/// container for all data that are used by the unit
TYPE HandlingDataRef :
STRUCT
  Config : REFERENCE TO HandlingDataConfig; // data required for booting the unit (axes configuration, simulation, parameters that have to be written in PREOP, ...)
  Machine : REFERENCE TO HandlingDataMachine; // speeds, positions, ...
  Calibration : REFERENCE TO HandlingDataCalibration; // offsets, shifts of nominal to actual values
END_STRUCT
END_TYPE

(* stored: Version 1.1.0.1
   DUT HandlingDataRef: Id {ec23e898-337f-470f-ad58-2e15c8da0680} *)
